Yaskawa INFORM job: KRIS1(-160_-90)07.JBI

/JOB
//NAME KRIS1(-160_-90)07
//POS
///NPOS 270,270,270,15,0,0
///TOOL 0
///POSTYPE PULSE
///PULSE
C00000=1357,-104031,-113776,-9484,62521,-80538
C00001=1357,-104031,-113776,-9484,62521,-80538
C00002=36470,-76528,-106815,-19279,71473,-77234
C00003=134470,-76528,-106815,-19279,71473,-77234
C00004=174981,-50493,-90161,-40064,84672,-66854
C00005=187879,-63712,-94262,-49080,81916,-61249
C00006=186060,-71155,-91964,-59790,82905,-66762
C00007=178869,-72848,-88692,-57971,77164,-66872
C00008=178869,-73293,-87273,-58169,76560,-66435
C00009=178869,-73560,-86246,-58315,76140,-66130
C00010=178674,-73111,-86205,-58218,76137,-66246
C00011=177360,-70267,-84836,-57702,75706,-66732
C00012=178674,-73111,-86205,-58218,76137,-66246
C00013=178674,-71838,-89995,-57689,77779,-67427
C00014=187879,-63712,-94262,-49080,81916,-61249
C00015=188382,-49930,-83952,-49213,82654,-61403
C00016=188014,-50962,-81654,-49243,81175,-60803
C00017=188014,-51673,-80691,-49342,80537,-60470
C00018=188014,-51583,-80818,-49329,80620,-60513
C00019=186548,-48975,-79328,-48719,80176,-60967
C00020=188014,-51583,-80818,-49329,80620,-60513
C00021=188014,-47372,-85350,-48920,83933,-62231
C00022=182062,-62332,-92296,-30199,64588,-50507
C00023=184090,-61700,-84500,-30217,57788,-46513
C00024=184090,-62275,-83323,-30540,56902,-46238
C00025=184090,-62207,-83473,-30499,57013,-46272
C00026=182547,-59219,-81900,-29317,56990,-46927
C00027=184090,-62207,-83473,-30499,57013,-46272
C00028=182062,-62332,-92296,-30199,64588,-50507
C00029=213458,-81436,-127572,-45024,85737,-46387
C00030=213462,-137262,-127618,-80891,60645,-46377
C00031=213462,-137262,-127618,-80891,60645,-46377
C00032=213462,-137262,-127281,-45256,60365,-46369
C00033=190178,-104312,-111371,-30656,55898,-55861
C00034=182510,-123951,-113302,-29184,45443,-56133
C00035=182510,-123446,-111392,-29630,44641,-55847
C00036=182510,-123495,-111565,-29589,44713,-55873
C00037=180510,-119420,-110276,-27514,45182,-57098
C00038=182510,-123495,-111565,-29589,44713,-55873
C00039=182510,-124409,-115363,-28705,46354,-56443
C00040=219776,-105077,-106077,-50090,64862,-45838
C00041=220601,-99189,-101769,-50266,65553,-45786
C00042=220601,-99263,-100237,-50600,64914,-45410
C00043=220601,-99258,-100424,-50559,64990,-45455
C00044=218392,-97957,-99927,-49618,64034,-46123
C00045=220601,-99258,-100424,-50559,64990,-45455
C00046=219776,-105077,-106077,-50090,64862,-45838
C00047=190178,-104312,-111371,-30656,55898,-55861
C00048=229240,-109114,-135810,-47014,82062,-49329
C00049=229240,-109114,-135810,-47014,82062,-49329
C00050=195224,-66819,-119592,-28790,78815,-60275
C00051=159578,-94739,-111578,-14965,102577,-71346
C00052=157566,-87256,-71357,-3912,80960,-68626
C00053=158237,-87274,-67249,-3997,78461,-68317
C00054=158512,-86753,-64553,-4040,77085,-68177
C00055=158512,-85902,-62577,-4050,76306,-68151
C00056=159334,-88042,-63583,-4126,75872,-67853
C00057=159947,-89575,-64280,-4185,75546,-67628
C00058=158678,-86897,-63962,-4060,76658,-68106
C00059=158401,-87046,-65688,-4022,77628,-68233
C00060=157724,-87159,-69865,-3934,80101,-68545
C00061=157573,-90681,-89077,-3900,90084,-68907
C00062=157703,-92030,-92713,-3898,91631,-68910
C00063=158377,-93978,-89476,-3949,88678,-68591
C00064=158653,-94353,-86922,-3974,86930,-68442
C00065=158653,-94065,-85585,-3975,86257,-68419
C00066=158901,-94897,-86117,-3998,86172,-68332
C00067=159738,-97484,-87119,-4071,85502,-68025
C00068=158508,-94414,-86637,-3961,86718,-68485
C00069=158233,-93872,-88035,-3937,87841,-68614
C00070=157561,-92106,-91348,-3883,90748,-68930
C00071=157550,-88189,-103730,-3988,100358,-69239
C00072=157494,-88262,-105997,-3987,101710,-69297
C00073=158163,-92718,-103752,-3992,98079,-68960
C00074=158927,-96366,-102620,-4029,95553,-68625
C00075=158927,-96520,-101690,-4026,94903,-68601
C00076=158927,-96495,-101852,-4026,95015,-68605
C00077=159979,-100458,-103367,-4107,93966,-68220
C00078=158702,-95424,-101809,-4010,95525,-68699
C00079=158425,-94019,-102865,-4000,96880,-68834
C00080=157748,-89886,-105246,-3989,100429,-69172
C00081=156260,-82084,-105550,-20461,72444,-69801
C00082=137260,-84248,-120477,-10166,77039,-76482
C00083=137260,-138866,-133764,-10166,31487,-76482
C00084=72641,-154229,-133982,-11252,19318,-75992
C00085=56453,-149109,-122299,-13274,13706,-75060
C00086=30023,-158112,-125301,-6799,9035,-78029
C00087=-11401,-148032,-125425,-11667,35640,-75771
C00088=-126225,-114648,-117375,-36487,17100,-65054
C00089=-160935,-140983,-109640,-13468,75088,-74332
C00090=-169853,-118963,-84593,-12681,69660,86771
C00091=-185015,-85467,-64977,-10138,72568,81037
C00092=-186046,-86587,-63372,-10054,70902,80807
C00093=-186046,-85672,-61299,-10100,70108,80875
C00094=-186099,-85805,-61481,-10085,70145,80849
C00095=-187639,-87511,-62050,-9863,69435,80354
C00096=-183812,-88241,-67244,-10331,72692,81455
C00097=-173907,-109296,-96285,-11524,80966,84205
C00098=-165243,-81442,-84446,-9619,88683,83239
C00099=-165243,-81286,-81084,-9622,86723,83389
C00100=-165344,-81527,-80785,-9608,86408,83377
C00101=-165344,-81401,-79599,-9612,85752,83428
C00102=-165344,-81434,-79892,-9611,85913,83415
C00103=-166373,-84175,-81092,-9484,85132,83124
C00104=-163979,-82682,-81772,-9785,86585,83830
C00105=-160654,-84295,-101618,-10197,98198,83833
C00106=-158831,-94543,-102742,-7696,93888,81952
C00107=-159073,-94488,-101668,-7659,93239,81911
C00108=-159073,-94700,-100523,-7653,92432,81960
C00109=-159073,-94669,-100714,-7655,92565,81952
C00110=-160071,-98397,-102165,-7522,91459,81686
C00111=-158831,-94357,-103427,-7703,94400,81921
C00112=-161715,-86803,-103327,-4886,98608,77730
C00113=-162141,-92472,-85533,3463,86932,68770
C00114=-161818,-87798,-71417,3733,80713,68419
C00115=-160875,-83714,-65601,3665,79192,68698
C00116=-161375,-83882,-63363,3725,77755,68482
C00117=-161375,-83186,-61665,3733,77069,68462
C00118=-161375,-83302,-61946,3731,77181,68466
C00119=-162606,-86103,-62964,3849,76427,68017
C00120=-161375,-84160,-64056,3722,78038,68491
C00121=-162005,-87841,-70029,3758,79847,68329
C00122=-161949,-92223,-96357,3744,93768,68761
C00123=-161804,-92637,-92737,3704,91325,68737
C00124=-160782,-89227,-87327,3611,89709,69033
C00125=-161425,-90912,-85851,3665,87970,68764
C00126=-161425,-90690,-84578,3665,87303,68744
C00127=-161425,-90728,-84781,3665,87408,68747
C00128=-162412,-93603,-85938,3751,86691,68391
C00129=-161425,-91016,-86520,3665,88326,68774
C00130=-162058,-93372,-91608,3722,90267,68620
C00131=-162002,-88104,-107646,3859,102814,69021
C00132=-161873,-89540,-106233,3806,101205,69011
C00133=-162580,-93883,-103932,3818,97597,68666
C00134=-159915,-93477,-102438,3577,96772,69526
C00135=-159915,-93839,-100899,3567,95642,69493
C00136=-159915,-93799,-101099,3568,95785,69497
C00137=-160794,-97042,-102371,3639,94941,69180
C00138=-159915,-93165,-103472,3585,97568,69550
C00139=-164885,-102201,-108421,4002,96197,67859
C00140=-149595,-96211,-103761,5489,101844,74102
C00141=-148895,-100989,-103442,6283,96942,74202
C00142=-149006,-93113,-100988,5479,101691,74295
C00143=-149599,-96300,-103483,5484,101628,74092
C00144=-137295,-108190,-106060,5698,94014,77976
C00145=-149608,-96287,-103789,5489,101823,74097
C00146=-160720,-151449,-123129,13814,72249,68439
C00147=-174899,-138237,-126795,-1008,88740,67536
C00148=-163022,-96341,-102515,-22398,105363,76518
C00149=-163017,-96713,-99258,-22147,103326,76913
C00150=-166118,-105377,-102170,-18852,96347,77230
C00151=-163022,-96736,-99152,-22139,103253,76925
C00152=-162158,-93804,-96763,-22109,103515,77196
C00153=-174925,-92085,-97088,-18785,97864,73864
C00154=-167549,-101389,-103915,-18999,98984,76305
C00155=-163194,-119427,-113025,-19710,97619,78016
C00156=-163006,-95534,-87485,-21597,97146,78065
C00157=-166449,-103981,-88986,-17839,88165,78380
C00158=-167279,-118842,-91930,-16839,77497,71410
C00159=-163006,-94576,-83573,-21494,95359,78388
C00160=-162142,-91714,-81191,-21448,95589,78662
C00161=-178049,-105864,-87645,-15594,79224,67328
C00162=-171906,-113065,-93299,-16245,80217,69386
C00163=-173072,-122981,-101575,4997,88706,65554
C00164=-166636,-106884,-92426,2568,94448,67910
C00165=-167630,-109607,-91139,2502,92292,67531
C00166=-162194,-92631,-84353,-657,102863,69400
C00167=-163060,-95514,-86735,-782,102839,69097
C00168=-155875,-120106,-94474,3152,88541,71437
C00169=-155875,-121766,-97691,3153,89666,71465
C00170=-178442,-133591,-104623,8068,82135,63325
C00171=-176542,-133362,-109369,6755,86992,64211
C00172=-163036,-88875,-67291,-2288,96831,69180
C00173=-159610,-85618,-62441,-1680,95605,70370
C00174=-162086,-85813,-60042,-2106,93969,69554
C00175=-162173,-84225,-60457,-2128,95039,69506
C00176=-163038,-86971,-62872,-2279,95091,69211
C00177=-151835,-92381,-62525,-304,92274,73022
C00178=-151835,-95702,-69255,-305,94709,73016
C00179=-163041,-94022,-81579,-12660,98605,75478
C00180=-162985,-87715,-64806,-21312,87868,79725
C00181=-162980,-85781,-60474,-21324,86307,80003
C00182=-163244,-83528,-57038,-21357,85347,80079
C00183=-162985,-85725,-60330,-21325,86250,80011
C00184=-162122,-82990,-57905,-21265,86391,80297
C00185=-171549,-75890,-53739,-21771,84944,77151
C00186=-153122,-94015,-66237,-20488,88162,83220
C00187=-168603,-127327,-105850,-12339,78437,-77405
C00188=-149894,-144724,-110594,-14594,75698,-70467
C00189=-126225,-114648,-117375,-36487,17100,-65054
C00190=-118781,-153853,-134406,-32592,23357,-65054
C00191=-12470,-167083,-125425,-11667,16324,-75771
C00192=137258,-84249,-120477,-10166,64820,-76482
C00193=160540,-100857,-113063,-23155,68829,-67581
C00194=174981,-50493,-90161,-40064,84672,-66854
C00195=187879,-63712,-94262,-49080,81916,-61249
C00196=230671,-89591,-126680,-64018,108053,-56526
C00197=230671,-150117,-126680,-83924,107200,-56526
C00198=230671,-150117,-126680,-83924,107200,-56526
C00199=230671,-150117,-126680,-39809,88276,-56526
C00200=185677,-128245,-133585,-38839,68006,-71149
C00201=143279,-154007,-127386,-2438,36675,-82296
C00202=143641,-141701,-120251,-2678,38614,-82167
C00203=143742,-142485,-120562,-2786,38406,-82105
C00204=143590,-141570,-120589,-2614,38886,-82201
C00205=202481,-119765,-113580,-40189,62069,-59692
C00206=198646,-130340,-109614,-41067,39992,-50520
C00207=196873,-131559,-103686,-47690,28279,-43258
C00208=193242,-140218,-107458,-47365,24899,-43542
C00209=143279,-154007,-127386,-2438,36675,-82296
C00210=143372,-162538,-136969,-2444,38193,-82294
C00211=143372,-162538,-136969,-2444,38193,-82294
C00212=169193,-120980,-126540,-32650,66176,-77929
C00213=162706,-113692,-115443,-30259,61179,-79142
C00214=159752,-104020,-109361,-28408,61247,-80415
C00215=143742,-142485,-120562,-2786,38406,-82105
C00216=143590,-141570,-120589,-2614,38886,-82201
C00217=133258,-125438,-116737,-13449,48460,-89137
C00218=140125,-121566,-112050,-33225,52073,-88232
C00219=147500,-115752,-104174,-50028,56665,-87600
C00220=148531,-114571,-100134,-56979,57308,-87783
C00221=151078,-112408,-101145,-56872,59820,-87990
C00222=162706,-113692,-115443,-30259,61179,-79142
C00223=169193,-120980,-126540,-32650,66176,-77929
C00224=169193,-120980,-126540,-32650,66176,-77929
C00225=169193,-120980,-126540,-32650,66176,-77929
C00226=169193,-120980,-126540,-32650,66176,-77929
C00227=189746,-144194,-133392,-42604,68859,-69788
C00228=182215,-131283,-122466,-40105,65254,-71827
C00229=178274,-121415,-115340,-38427,64020,-73174
C00230=157461,-154213,-124395,-33339,46072,-76518
C00231=155749,-154222,-121631,-44079,49487,-78540
C00232=159534,-158630,-125101,-47522,52653,-77846
C00233=179897,-166210,-133900,-51769,64813,-73191
C00234=179897,-166210,-133900,-51769,64813,-73191
C00235=179897,-166210,-133900,-51769,64813,-73191
C00236=144017,-127352,-123370,-33815,56946,-88116
C00237=136296,-120281,-120593,4079,55650,-85264
C00238=135299,-107675,-113640,4618,57894,-85562
C00239=145232,-101484,-111409,-1707,59530,-81793
C00240=158760,-87446,-105850,-9753,64232,-77140
C00241=147394,-98337,-102183,17301,47751,-78343
C00242=144875,-102905,-108473,14295,50590,-79740
C00243=136296,-120281,-120593,4079,55650,-85264
C00244=138675,-113827,-131364,2561,67962,-83610
C00245=184171,-107868,-119248,-16468,98370,-62097
C00246=171634,-136713,-119987,-14813,82155,-64373
C00247=159470,-98078,-104776,-5796,102446,-69552
C00248=161378,-95420,-100865,-5759,101546,-68862
C00249=158743,-95268,-103371,-5812,102972,-69826
C00250=157888,-92366,-100981,-5813,102933,-70115
C00251=150653,-106168,-104972,-5675,97814,-72341
C00252=153886,-106740,-107354,-5718,99208,-71304
C00253=163031,-143044,-118600,-5591,88166,-67691
C00254=166711,-113552,-95038,-4166,94777,-66107
C00255=166288,-102352,-87247,-1195,97977,-66532
C00256=158755,-94787,-86481,976,103949,-69303
C00257=157900,-91912,-84097,841,103969,-69603
C00258=155716,-111746,-90511,-2417,94923,-70111
C00259=153517,-115912,-96262,-2679,96250,-70891
C00260=166250,-149525,-105399,-1185,84912,-66421
C00261=160517,-92560,-68375,-1999,97708,-69937
C00262=161332,-84623,-58779,-1824,95900,-69631
C00263=158782,-86330,-62292,-2348,97119,-70521
C00264=157926,-83586,-59872,-2521,97014,-70811
C00265=150683,-91270,-61306,-3946,93662,-73181
C00266=149643,-98229,-74267,-4194,97999,-73676
C00267=159578,-94739,-111578,-14965,102577,-71346
C00268=134470,-76528,-106815,-19279,71473,-77234
C00269=36470,-76528,-106815,-19279,71473,-77234
BC00000=230661,511423,1075115
BC00001=230661,511423,1075115
BC00002=295309,515546,1075139
BC00003=353519,294132,1075139
BC00004=353008,251675,1075139
BC00005=352559,214443,1075139
BC00006=352563,214698,1075132
BC00007=352563,214698,1075132
BC00008=352563,214698,1075132
BC00009=352563,214698,1075132
BC00010=352563,214698,1075132
BC00011=352563,214698,1075132
BC00012=352563,214698,1075132
BC00013=352563,214698,1075132
BC00014=352559,214443,1075139
BC00015=352559,214443,1075139
BC00016=352559,214443,1075139
BC00017=352559,214443,1075139
BC00018=352559,214443,1075139
BC00019=352559,214443,1075136
BC00020=352559,214443,1075139
BC00021=352559,214443,1075139
BC00022=352559,214443,1075135
BC00023=352559,214443,1075135
BC00024=352559,214443,1075135
BC00025=352559,214443,1075135
BC00026=352559,214443,1075135
BC00027=352559,214443,1075135
BC00028=352559,214443,1075135
BC00029=352559,214443,1075135
BC00030=352559,214443,1075135
BC00031=265654,200751,1075135
BC00032=265654,200751,1075135
BC00033=265654,182191,1075135
BC00034=265654,182191,1075135
BC00035=265654,182191,1075135
BC00036=265654,182191,1075135
BC00037=265654,182191,1075135
BC00038=265654,182191,1075135
BC00039=265654,182191,1075135
BC00040=265654,153562,1075135
BC00041=265654,153562,1075135
BC00042=265654,153562,1075135
BC00043=265654,153562,1075135
BC00044=265654,153562,1075135
BC00045=265654,153562,1075135
BC00046=265654,153562,1075135
BC00047=265654,182191,1075135
BC00048=288097,183452,1075134
BC00049=288097,183452,1075134
BC00050=366407,228141,1075134
BC00051=353519,214242,1075139
BC00052=382934,213120,1075139
BC00053=382934,213120,1075139
BC00054=382934,213120,1075139
BC00055=382934,213120,1075139
BC00056=382933,213121,1075138
BC00057=382933,213121,1075138
BC00058=382934,213120,1075139
BC00059=382934,213120,1075139
BC00060=382934,213120,1075139
BC00061=382615,202068,1075139
BC00062=382076,183746,1075139
BC00063=382076,183746,1075139
BC00064=382076,183746,1075139
BC00065=382076,183746,1075139
BC00066=382076,183746,1075139
BC00067=382076,183746,1075139
BC00068=382076,183746,1075139
BC00069=382076,183746,1075139
BC00070=382076,183746,1075139
BC00071=382031,172700,1075139
BC00072=382054,156718,1075139
BC00073=382054,156718,1075139
BC00074=382054,156718,1075139
BC00075=382054,156718,1075139
BC00076=382054,156718,1075139
BC00077=382054,156718,1075139
BC00078=382054,156718,1075139
BC00079=382054,156718,1075139
BC00080=382054,156718,1075139
BC00081=381880,223521,1075139
BC00082=353800,266120,1075139
BC00083=353800,266120,1075139
BC00084=369629,142690,1075139
BC00085=373603,111702,1075139
BC00086=379757,63718,1075139
BC00087=398174,159824,1075139
BC00088=312616,52052,1075139
BC00089=340737,74809,1075139
BC00090=340750,75261,1075139
BC00091=340750,75261,1075139
BC00092=340750,75261,1075139
BC00093=340750,75261,1075139
BC00094=340750,75261,1075139
BC00095=340750,75261,1075139
BC00096=340750,75261,1075139
BC00097=340750,75261,1075139
BC00098=322858,75822,1075139
BC00099=322858,75822,1075139
BC00100=322858,75822,1075139
BC00101=322858,75822,1075139
BC00102=322858,75822,1075139
BC00103=322858,75822,1075139
BC00104=322858,75822,1075139
BC00105=321852,75909,1075139
BC00106=305307,104079,1075139
BC00107=305307,104079,1075139
BC00108=305307,104079,1075139
BC00109=305307,104079,1075139
BC00110=305307,104079,1075139
BC00111=305307,104079,1075139
BC00112=323389,89421,1075139
BC00113=381448,44122,1075139
BC00114=383279,43102,1075139
BC00115=383279,43102,1075139
BC00116=383279,43102,1075139
BC00117=383279,43102,1075139
BC00118=383279,43102,1075139
BC00119=383279,43102,1075139
BC00120=383279,43102,1075139
BC00121=383279,43102,1075139
BC00122=383346,62866,1075139
BC00123=383236,72913,1075139
BC00124=383236,72913,1075139
BC00125=383236,72913,1075139
BC00126=383236,72913,1075139
BC00127=383236,72913,1075139
BC00128=383236,72913,1075139
BC00129=383236,72913,1075139
BC00130=383236,72913,1075139
BC00131=383192,91135,1075139
BC00132=383033,99727,1075139
BC00133=383033,99727,1075139
BC00134=383033,99727,1075139
BC00135=383033,99727,1075139
BC00136=383033,99727,1075139
BC00137=383033,99727,1075139
BC00138=383033,99727,1075139
BC00139=383033,99727,1075139
BC00140=348621,100905,1075139
BC00141=348896,99875,1075139
BC00142=348896,99875,1075139
BC00143=348896,99875,1075139
BC00144=348896,99875,1075139
BC00145=364549,100867,1075139
BC00146=363863,103441,1075139
BC00147=346080,121643,1075139
BC00148=323509,144746,1075139
BC00149=322803,140398,1075139
BC00150=322592,139099,1075139
BC00151=322520,138659,1075139
BC00152=322520,138659,1075139
BC00153=322592,139099,1075139
BC00154=322592,139099,1075139
BC00155=318216,140757,1075139
BC00156=323435,117945,1075139
BC00157=322729,113597,1075139
BC00158=322729,113597,1075139
BC00159=322446,111858,1075139
BC00160=322446,111858,1075139
BC00161=322729,113597,1075139
BC00162=322729,113597,1075139
BC00163=364623,109054,1075139
BC00164=365306,105037,1075139
BC00165=365306,105037,1075139
BC00166=365579,103431,1075139
BC00167=365579,103431,1075139
BC00168=365306,105037,1075139
BC00169=365306,105037,1075139
BC00170=380551,109015,1075139
BC00171=378551,106052,1075139
BC00172=364555,85312,1075139
BC00173=365237,80960,1075139
BC00174=365237,80960,1075139
BC00175=365509,79219,1075139
BC00176=365509,79219,1075139
BC00177=365237,80960,1075139
BC00178=365237,80960,1075139
BC00179=341067,86785,1075139
BC00180=323352,88165,1075139
BC00181=322645,83817,1075139
BC00182=322645,83817,1075139
BC00183=322363,82077,1075139
BC00184=322363,82077,1075139
BC00185=322645,83817,1075139
BC00186=306969,83854,1075139
BC00187=340737,74809,1075139
BC00188=340737,74809,1075139
BC00189=312616,52052,1075139
BC00190=312616,52052,1075139
BC00191=398174,159824,1075139
BC00192=353801,266119,1075139
BC00193=381880,223521,1075139
BC00194=353008,251675,1075139
BC00195=352559,214443,1075139
BC00196=352559,214443,1075139
BC00197=269474,214443,1075139
BC00198=209500,192764,1075139
BC00199=229937,192764,1075139
BC00200=209500,192764,1075139
BC00201=209500,192764,1075139
BC00202=209500,192764,1075135
BC00203=209500,192764,1075135
BC00204=209500,192764,1075135
BC00205=234557,161453,1075132
BC00206=234557,161453,1075132
BC00207=234557,161453,1075132
BC00208=234557,161453,1075132
BC00209=209500,192764,1075139
BC00210=209501,302299,1075135
BC00211=304046,302299,1075135
BC00212=304046,203195,1075135
BC00213=304046,203195,1075135
BC00214=304046,203195,1075135
BC00215=209500,192764,1075135
BC00216=209500,192764,1075135
BC00217=304046,203195,1075135
BC00218=304046,203195,1075135
BC00219=304046,203195,1075135
BC00220=304046,203195,1075135
BC00221=304046,203195,1075135
BC00222=304046,203195,1075135
BC00223=304046,203195,1075135
BC00224=304046,310775,1075135
BC00225=206063,312405,1075135
BC00226=206063,203684,1075135
BC00227=216899,182662,1075135
BC00228=216899,182662,1075135
BC00229=216899,182662,1075135
BC00230=216899,182662,1075135
BC00231=216898,182663,1075134
BC00232=216899,182662,1075135
BC00233=216898,182662,1075132
BC00234=216898,281603,1075132
BC00235=299601,281603,1075132
BC00236=274761,236253,1075132
BC00237=304046,203195,1075135
BC00238=304046,203195,1075135
BC00239=304046,203195,1075135
BC00240=304045,203195,1075131
BC00241=304046,203195,1075135
BC00242=304046,203195,1075135
BC00243=304046,203195,1075135
BC00244=308056,199315,1075135
BC00245=363620,145544,1075139
BC00246=363620,145544,1075139
BC00247=364348,148086,1075139
BC00248=364638,149103,1075136
BC00249=364639,149103,1075139
BC00250=364639,149103,1075139
BC00251=364638,149103,1075136
BC00252=370099,148733,1075137
BC00253=370099,148733,1075137
BC00254=364145,147610,1075137
BC00255=364418,149141,1075138
BC00256=364758,151053,1075139
BC00257=364758,151053,1075139
BC00258=364418,149141,1075138
BC00259=364418,149141,1075138
BC00260=364418,149141,1075138
BC00261=353519,171684,1075139
BC00262=355504,177664,1075139
BC00263=355504,177664,1075139
BC00264=355504,177664,1075139
BC00265=355504,177664,1075139
BC00266=355504,177664,1075139
BC00267=353519,214242,1075139
BC00268=353519,294132,1075139
BC00269=295309,515546,1075139
EC00000=-12352,-159808
EC00001=1418783,-184756
EC00002=1418945,372643
EC00003=1418945,372643
EC00004=1342906,372643
EC00005=1276223,372643
EC00006=1276676,372643
EC00007=1276676,372643
EC00008=1276676,372643
EC00009=1276676,372643
EC00010=1276676,372643
EC00011=1276676,372643
EC00012=1276676,372643
EC00013=1276676,372643
EC00014=1276223,372643
EC00015=1276223,372643
EC00016=1276223,372643
EC00017=1276223,372643
EC00018=1276223,372643
EC00019=1276222,372643
EC00020=1276223,372643
EC00021=1276223,372643
EC00022=1276222,372644
EC00023=1276222,372644
EC00024=1276222,372644
EC00025=1276222,372644
EC00026=1276222,372644
EC00027=1276222,372644
EC00028=1276222,372644
EC00029=1276222,372644
EC00030=1276222,372644
EC00031=1276222,372644
EC00032=1276222,372644
EC00033=1276222,372644
EC00034=1276222,372644
EC00035=1276222,372644
EC00036=1276222,372644
EC00037=1276222,372644
EC00038=1276222,372644
EC00039=1276222,372644
EC00040=1276222,372644
EC00041=1276222,372644
EC00042=1276222,372644
EC00043=1276222,372644
EC00044=1276222,372644
EC00045=1276222,372644
EC00046=1276222,372644
EC00047=1276222,372644
EC00048=1276222,372644
EC00049=1276222,372644
EC00050=1276222,372644
EC00051=1418945,372643
EC00052=1418945,372643
EC00053=1418945,372643
EC00054=1418945,372643
EC00055=1418945,372643
EC00056=1418943,372643
EC00057=1418943,372643
EC00058=1418945,372643
EC00059=1418945,372643
EC00060=1418945,372643
EC00061=1418945,372643
EC00062=1418945,372643
EC00063=1418945,372643
EC00064=1418945,372643
EC00065=1418945,372643
EC00066=1418945,372643
EC00067=1418945,372643
EC00068=1418945,372643
EC00069=1418945,372643
EC00070=1418945,372643
EC00071=1418945,372643
EC00072=1418945,372643
EC00073=1418945,372643
EC00074=1418945,372643
EC00075=1418945,372643
EC00076=1418945,372643
EC00077=1418945,372643
EC00078=1418945,372643
EC00079=1418945,372643
EC00080=1418945,372643
EC00081=1418945,372643
EC00082=1418945,372643
EC00083=1418945,372643
EC00084=1418945,372643
EC00085=1418945,372643
EC00086=1418945,372643
EC00087=1595090,-179995
EC00088=1773681,-740307
EC00089=1773681,-740307
EC00090=1773681,-740307
EC00091=1773681,-740307
EC00092=1773681,-740307
EC00093=1773681,-740307
EC00094=1773681,-740307
EC00095=1773681,-740307
EC00096=1773681,-740307
EC00097=1773681,-740307
EC00098=1773681,-740307
EC00099=1773681,-740307
EC00100=1773681,-740307
EC00101=1773681,-740307
EC00102=1773681,-740307
EC00103=1773681,-740307
EC00104=1773681,-740307
EC00105=1773681,-740307
EC00106=1773681,-740307
EC00107=1773681,-740307
EC00108=1773681,-740307
EC00109=1773681,-740307
EC00110=1773681,-740307
EC00111=1773681,-740307
EC00112=1773681,-740307
EC00113=1773681,-740307
EC00114=1773681,-740307
EC00115=1773681,-740307
EC00116=1773681,-740307
EC00117=1773681,-740307
EC00118=1773681,-740307
EC00119=1773681,-740307
EC00120=1773681,-740307
EC00121=1773681,-740307
EC00122=1773681,-740307
EC00123=1773681,-740307
EC00124=1773681,-740307
EC00125=1773681,-740307
EC00126=1773681,-740307
EC00127=1773681,-740307
EC00128=1773681,-740307
EC00129=1773681,-740307
EC00130=1773681,-740307
EC00131=1773681,-740307
EC00132=1773681,-740307
EC00133=1773681,-740307
EC00134=1773681,-740307
EC00135=1773681,-740307
EC00136=1773681,-740307
EC00137=1773681,-740307
EC00138=1773681,-740307
EC00139=1773681,-740307
EC00140=1773681,-740307
EC00141=1773681,-740307
EC00142=1773681,-740307
EC00143=1773681,-740307
EC00144=1773681,-740307
EC00145=1773681,-740307
EC00146=1773681,-740307
EC00147=1773681,-740307
EC00148=1773681,-740307
EC00149=1773681,-740307
EC00150=1773681,-740307
EC00151=1773681,-740307
EC00152=1773681,-740307
EC00153=1773681,-740307
EC00154=1773681,-740307
EC00155=1773681,-740307
EC00156=1773681,-740307
EC00157=1773681,-740307
EC00158=1773681,-740307
EC00159=1773681,-740307
EC00160=1773681,-740307
EC00161=1773681,-740307
EC00162=1773681,-740307
EC00163=1773681,-740307
EC00164=1773681,-740307
EC00165=1773681,-740307
EC00166=1773681,-740307
EC00167=1773681,-740307
EC00168=1773681,-740307
EC00169=1773681,-740307
EC00170=1773681,-740307
EC00171=1773681,-740307
EC00172=1773681,-740307
EC00173=1773681,-740307
EC00174=1773681,-740307
EC00175=1773681,-740307
EC00176=1773681,-740307
EC00177=1773681,-740307
EC00178=1773681,-740307
EC00179=1773681,-740307
EC00180=1773681,-740307
EC00181=1773681,-740307
EC00182=1773681,-740307
EC00183=1773681,-740307
EC00184=1773681,-740307
EC00185=1773681,-740307
EC00186=1773681,-740307
EC00187=1773681,-740307
EC00188=1773681,-740307
EC00189=1773681,-740307
EC00190=1773681,-740307
EC00191=1595090,-179995
EC00192=1418947,372636
EC00193=1418945,372643
EC00194=1342906,372643
EC00195=1276223,372643
EC00196=1276223,372643
EC00197=1276223,372643
EC00198=1276223,372643
EC00199=1276223,372643
EC00200=1276223,372643
EC00201=1276223,372643
EC00202=1276222,372643
EC00203=1276222,372643
EC00204=1276222,372643
EC00205=1276221,372643
EC00206=1276221,372643
EC00207=1276221,372643
EC00208=1276221,372643
EC00209=1276223,372643
EC00210=1276222,372643
EC00211=1276222,372643
EC00212=1276222,372643
EC00213=1276222,372643
EC00214=1276222,372643
EC00215=1276222,372643
EC00216=1276222,372643
EC00217=1276222,372643
EC00218=1276222,372643
EC00219=1276222,372643
EC00220=1276222,372643
EC00221=1276222,372643
EC00222=1276222,372643
EC00223=1276222,372643
EC00224=1276222,372643
EC00225=1276222,372643
EC00226=1276222,372643
EC00227=1276222,372643
EC00228=1276222,372643
EC00229=1276222,372643
EC00230=1276222,372643
EC00231=1276221,372644
EC00232=1276222,372643
EC00233=1276221,372643
EC00234=1276221,372643
EC00235=1276221,372643
EC00236=1276221,372643
EC00237=1276222,372643
EC00238=1276222,372643
EC00239=1276222,372643
EC00240=1276222,372644
EC00241=1276222,372643
EC00242=1276222,372643
EC00243=1276222,372643
EC00244=1285829,372643
EC00245=1418945,372643
EC00246=1418945,372643
EC00247=1418945,372643
EC00248=1418945,372643
EC00249=1418945,372643
EC00250=1418945,372643
EC00251=1418945,372643
EC00252=1418945,372643
EC00253=1418945,372643
EC00254=1418944,372643
EC00255=1418944,372643
EC00256=1418945,372643
EC00257=1418945,372643
EC00258=1418944,372643
EC00259=1418944,372643
EC00260=1418944,372643
EC00261=1418945,372643
EC00262=1418945,372643
EC00263=1418945,372643
EC00264=1418945,372643
EC00265=1418945,372643
EC00266=1418945,372643
EC00267=1418945,372643
EC00268=1418945,372643
EC00269=1418945,372643
///POSTYPE BASE
///RECTAN
///RCONF 0,0,0,0,1,0,0,0,0,0,0,0,0,0,0,0,0,0,0,0,0,0,0,0
P00006=2.006,1.622,-0.565,0.0000,0.0000,0.0000
P00021=0.073,2.058,-0.109,0.0000,0.0000,0.0000
P00022=2.006,1.622,-0.565,0.0000,0.0000,0.0000
///RCONF 0,0,0,0,0,0,0,0,0,0,0,0,0,0,0,0,0,0,0,0,0,0,0,0
P00023=-2.957,-4.083,2.762,0.0000,0.0000,0.0000
P00031=-0.170,0.039,-0.647,0.0000,0.0000,0.0000
P00032=-0.423,0.157,3.222,0.0000,0.0000,0.0000
P00033=0.854,-1.099,3.047,0.0000,0.0000,0.0000
///RCONF 0,0,0,0,1,0,0,0,0,0,0,0,0,0,0,0,0,0,0,0,0,0,0,0
P00034=-8.151,9.743,-4.393,0.0000,0.0000,0.0000
///RCONF 0,0,0,0,0,0,0,0,0,0,0,0,0,0,0,0,0,0,0,0,0,0,0,0
P00035=0.390,-0.027,1.040,0.0000,0.0000,0.0000
P00036=-2.434,0.084,0.197,0.0000,0.0000,0.0000
P00051=-5.945,4.696,-10.293,0.0000,0.0000,0.0000
P00052=-0.153,5.586,-7.982,0.0000,0.0000,0.0000
P00053=0.015,-0.644,-4.942,0.0000,0.0000,0.0000
P00054=-0.184,15.039,-0.270,0.0000,0.0000,0.0000
P00055=-0.009,2.790,-4.790,0.0000,0.0000,0.0000
//INST
///DATE 2024/11/18 15:49
///ATTR SC,RW
///GROUP1 RB1,BS1
///GROUP2 ST1
NOP
SFTOF
SSFTOF
SFTOF3D
'OK_r2_O7.1(P)(-160.-90)
MOVJ C00000 BC00000 VJ=100.00  +MOVJ EC00000 VJ=100.00
MOVJ C00001 BC00001 VJ=100.00  +MOVJ EC00001 VJ=100.00
MOVJ C00002 BC00002 VJ=100.00  +MOVJ EC00002 VJ=100.00
MOVJ C00003 BC00003 VJ=100.00  +MOVJ EC00003 VJ=100.00
MOVJ C00004 BC00004 VJ=50.00  +MOVJ EC00004 VJ=50.00
MOVJ C00005 BC00005 VJ=50.00  +MOVJ EC00005 VJ=50.00
'DODAC SEARCH NO NOWA SPOINE
MOVL C00006 BC00006 V=400.0  +MOVJ EC00006 VJ=100.00
SMOVL C00007 BC00007 V=400.0  +MOVJ EC00007
SFTOF3D
SMOVL C00008 BC00008 V=100.0  +MOVJ EC00008
SREFP 3 C00009 BC00009  +REFP EC00009
CALL JOB:SEARCH-R1-S13D
SET P051 P006
SFTON3D P051
SMOVL C00010 BC00010 V=100.0  +MOVJ EC00010
SREFP 3 C00011 BC00011  +REFP EC00011
CALL JOB:SEARCH-R1-S13D
SET P051 P006
SFTON3D P051
SMOVL C00012 BC00012 V=100.0  +MOVJ EC00012
MOVL C00013 BC00013 V=400.0  +MOVJ EC00013 VJ=100.00
MOVL C00014 BC00014 V=400.0  +MOVJ EC00014 VJ=100.00
SFTOF3D
MOVL C00015 BC00015 V=400.0  +MOVJ EC00015 VJ=100.00
SMOVL C00016 BC00016 V=100.0  +MOVJ EC00016
SREFP 3 C00017 BC00017  +REFP EC00017
CALL JOB:SEARCH-R1-S13D
SET P052 P006
SFTON3D P052
SMOVL C00018 BC00018 V=100.0  +MOVJ EC00018
SREFP 3 C00019 BC00019  +REFP EC00019
CALL JOB:SEARCH-R1-S13D
SET P052 P006
SFTON3D P052
SMOVL C00020 BC00020 V=100.0  +MOVJ EC00020
MOVL C00021 BC00021 V=400.0  +MOVJ EC00021 VJ=100.00
SFTOF3D
MOVL C00022 BC00022 V=400.0  +MOVJ EC00022 VJ=100.00
SMOVL C00023 BC00023 V=100.0  +MOVJ EC00023
SREFP 3 C00024 BC00024  +REFP EC00024
CALL JOB:SEARCH-R1-S13D
SET P053 P006
SFTON3D P053
SMOVL C00025 BC00025 V=100.0  +MOVJ EC00025
SREFP 3 C00026 BC00026  +REFP EC00026
CALL JOB:SEARCH-R1-S13D
SET P053 P006
SFTON3D P053
SMOVL C00027 BC00027 V=100.0  +MOVJ EC00027
MOVL C00028 BC00028 V=400.0  +MOVJ EC00028 VJ=100.00
SFTOF3D
MOVL C00029 BC00029 V=400.0  +MOVJ EC00029 VJ=100.00
MOVL C00030 BC00030 V=400.0  +MOVJ EC00030 VJ=100.00
MOVL C00031 BC00031 V=400.0  +MOVJ EC00031 VJ=100.00
MOVL C00032 BC00032 V=400.0  +MOVJ EC00032 VJ=100.00
SFTOF3D
MOVL C00033 BC00033 V=400.0  +MOVJ EC00033 VJ=100.00
SMOVL C00034 BC00034 V=100.0  +MOVJ EC00034
SREFP 3 C00035 BC00035  +REFP EC00035
CALL JOB:SEARCH-R1-S13D
SET P054 P006
SFTON3D P054
SMOVL C00036 BC00036 V=100.0  +MOVJ EC00036
SREFP 3 C00037 BC00037  +REFP EC00037
CALL JOB:SEARCH-R1-S13D
SET P054 P006
SFTON3D P054
SMOVL C00038 BC00038 V=100.0  +MOVJ EC00038
MOVL C00039 BC00039 V=400.0  +MOVJ EC00039 VJ=100.00
SFTOF3D
MOVL C00040 BC00040 V=400.0  +MOVJ EC00040 VJ=100.00
SMOVL C00041 BC00041 V=100.0  +MOVJ EC00041
SREFP 3 C00042 BC00042  +REFP EC00042
CALL JOB:SEARCH-R1-S13D
SET P055 P006
SFTON3D P055
SMOVL C00043 BC00043 V=100.0  +MOVJ EC00043
SREFP 3 C00044 BC00044  +REFP EC00044
CALL JOB:SEARCH-R1-S13D
SET P055 P006
SFTON3D P055
SMOVL C00045 BC00045 V=100.0  +MOVJ EC00045
MOVL C00046 BC00046 V=400.0  +MOVJ EC00046 VJ=100.00
SFTOF3D
MOVL C00047 BC00047 V=400.0  +MOVJ EC00047 VJ=100.00
MOVL C00048 BC00048 V=400.0  +MOVJ EC00048 VJ=100.00
MOVL C00049 BC00049 V=400.0  +MOVJ EC00049 VJ=100.00
MOVL C00050 BC00050 V=400.0  +MOVJ EC00050 VJ=100.00
MOVJ C00051 BC00051 VJ=100.00  +MOVJ EC00051 VJ=100.00
'Path S1422
SFTOF3D
MOVJ C00052 BC00052 VJ=100.00  +MOVJ EC00052 VJ=100.00
MOVL C00053 BC00053 V=400.0  +MOVJ EC00053 VJ=100.00
SMOVL C00054 BC00054 V=100.0  +MOVJ EC00054
SREFP 3 C00055 BC00055  +REFP EC00055
CALL JOB:SEARCH-R1-S13D
SET P021 P006
SFTON3D P021
SMOVL C00056 BC00056 V=100.0  +MOVJ EC00056
SREFP 3 C00057 BC00057  +REFP EC00057
CALL JOB:SEARCH-R1-S13D
SET P021 P006
SFTON3D P021
SMOVL C00058 BC00058 V=100.0  +MOVJ EC00058
MOVL C00059 BC00059 V=400.0  +MOVJ EC00059 VJ=100.00
MOVL C00060 BC00060 V=1000.0  +MOVJ EC00060 VJ=100.00
MOVJ C00061 BC00061 VJ=100.00  +MOVJ EC00061 VJ=100.00
'Path S1423
SFTOF3D
MOVJ C00062 BC00062 VJ=100.00  +MOVJ EC00062 VJ=100.00
MOVL C00063 BC00063 V=400.0  +MOVJ EC00063 VJ=100.00
SMOVL C00064 BC00064 V=100.0  +MOVJ EC00064
SREFP 3 C00065 BC00065  +REFP EC00065
CALL JOB:SEARCH-R1-S13D
SET P022 P006
SFTON3D P022
SMOVL C00066 BC00066 V=100.0  +MOVJ EC00066
SREFP 3 C00067 BC00067  +REFP EC00067
CALL JOB:SEARCH-R1-S13D
SET P022 P006
SFTON3D P022
SMOVL C00068 BC00068 V=100.0  +MOVJ EC00068
MOVL C00069 BC00069 V=400.0  +MOVJ EC00069 VJ=100.00
MOVL C00070 BC00070 V=1000.0  +MOVJ EC00070 VJ=100.00
MOVJ C00071 BC00071 VJ=100.00  +MOVJ EC00071 VJ=100.00
'Path S1424
SFTOF3D
MOVJ C00072 BC00072 VJ=100.00  +MOVJ EC00072 VJ=100.00
MOVL C00073 BC00073 V=400.0  +MOVJ EC00073 VJ=100.00
SMOVL C00074 BC00074 V=100.0  +MOVJ EC00074
SREFP 3 C00075 BC00075  +REFP EC00075
CALL JOB:SEARCH-R1-S13D
SET P023 P006
SFTON3D P023
SMOVL C00076 BC00076 V=100.0  +MOVJ EC00076
SREFP 3 C00077 BC00077  +REFP EC00077
CALL JOB:SEARCH-R1-S13D
SET P023 P006
SFTON3D P023
SFTOF3D
SMOVL C00078 BC00078 V=100.0  +MOVJ EC00078
MOVL C00079 BC00079 V=400.0  +MOVJ EC00079 VJ=100.00
MOVL C00080 BC00080 V=1000.0  +MOVJ EC00080 VJ=100.00
'obrot
MOVJ C00081 BC00081 VJ=100.00  +MOVJ EC00081 VJ=100.00
MOVJ C00082 BC00082 VJ=100.00  +MOVJ EC00082 VJ=100.00
MOVJ C00083 BC00083 VJ=100.00  +MOVJ EC00083 VJ=100.00
MOVJ C00084 BC00084 VJ=50.00  +MOVJ EC00084 VJ=50.00
MOVJ C00085 BC00085 VJ=50.00  +MOVJ EC00085 VJ=50.00
MOVJ C00086 BC00086 VJ=100.00  +MOVJ EC00086 VJ=100.00
MOVJ C00087 BC00087 VJ=100.00  +MOVJ EC00087 VJ=100.00
MOVJ C00088 BC00088 VJ=100.00  +MOVJ EC00088 VJ=100.00
MOVJ C00089 BC00089 VJ=100.00  +MOVJ EC00089 VJ=100.00
'Path S1077
SFTOF3D
MOVJ C00090 BC00090 VJ=100.00  +MOVJ EC00090 VJ=100.00
MOVL C00091 BC00091 V=400.0  +MOVJ EC00091 VJ=100.00
SMOVL C00092 BC00092 V=100.0  +MOVJ EC00092
SREFP 3 C00093 BC00093  +REFP EC00093
CALL JOB:SEARCH-R1-S13D
SET P031 P006
SFTON3D P031
SMOVL C00094 BC00094 V=100.0  +MOVJ EC00094
SREFP 3 C00095 BC00095  +REFP EC00095
CALL JOB:SEARCH-R1-S13D
SET P031 P006
SFTON3D P031
SMOVL C00096 BC00096 V=100.0  +MOVJ EC00096
MOVL C00097 BC00097 V=1000.0  +MOVJ EC00097 VJ=100.00
MOVJ C00098 BC00098 VJ=100.00  +MOVJ EC00098 VJ=100.00
'Path S1078
SFTOF3D
MOVL C00099 BC00099 V=400.0  +MOVJ EC00099 VJ=100.00
SMOVL C00100 BC00100 V=100.0  +MOVJ EC00100
SREFP 3 C00101 BC00101  +REFP EC00101
CALL JOB:SEARCH-R1-S13D
SET P032 P006
SFTON3D P032
SMOVL C00102 BC00102 V=100.0  +MOVJ EC00102
SREFP 3 C00103 BC00103  +REFP EC00103
CALL JOB:SEARCH-R1-S13D
SET P032 P006
SFTON3D P032
SMOVL C00104 BC00104 V=100.0  +MOVJ EC00104
MOVL C00105 BC00105 V=1000.0  +MOVJ EC00105 VJ=100.00
'Path S1079
SFTOF3D
MOVL C00106 BC00106 V=400.0  +MOVJ EC00106 VJ=100.00
SMOVL C00107 BC00107 V=100.0  +MOVJ EC00107
SREFP 3 C00108 BC00108  +REFP EC00108
CALL JOB:SEARCH-R1-S13D
SET P033 P006
SFTON3D P033
SMOVL C00109 BC00109 V=100.0  +MOVJ EC00109
SREFP 3 C00110 BC00110  +REFP EC00110
CALL JOB:SEARCH-R1-S13D
SET P033 P006
SFTON3D P033
SMOVL C00111 BC00111 V=100.0  +MOVJ EC00111
MOVJ C00112 BC00112 VJ=100.00  +MOVJ EC00112 VJ=100.00
MOVJ C00113 BC00113 VJ=100.00  +MOVJ EC00113 VJ=100.00
'Path S1080
SFTOF3D
MOVJ C00114 BC00114 VJ=100.00  +MOVJ EC00114 VJ=100.00
MOVL C00115 BC00115 V=400.0  +MOVJ EC00115 VJ=100.00
SMOVL C00116 BC00116 V=100.0  +MOVJ EC00116
SREFP 3 C00117 BC00117  +REFP EC00117
CALL JOB:SEARCH-R1-S13D
SET P034 P006
SFTON3D P034
SMOVL C00118 BC00118 V=100.0  +MOVJ EC00118
SREFP 3 C00119 BC00119  +REFP EC00119
CALL JOB:SEARCH-R1-S13D
SET P034 P006
SFTON3D P034
SMOVL C00120 BC00120 V=100.0  +MOVJ EC00120
MOVL C00121 BC00121 V=1000.0  +MOVJ EC00121 VJ=100.00
MOVJ C00122 BC00122 VJ=100.00  +MOVJ EC00122 VJ=100.00
'Path S1081
SFTOF3D
MOVJ C00123 BC00123 VJ=100.00  +MOVJ EC00123 VJ=100.00
MOVL C00124 BC00124 V=400.0  +MOVJ EC00124 VJ=100.00
SMOVL C00125 BC00125 V=100.0  +MOVJ EC00125
SREFP 3 C00126 BC00126  +REFP EC00126
CALL JOB:SEARCH-R1-S13D
SET P035 P006
SFTON3D P035
SMOVL C00127 BC00127 V=100.0  +MOVJ EC00127
SREFP 3 C00128 BC00128  +REFP EC00128
CALL JOB:SEARCH-R1-S13D
SET P035 P006
SFTON3D P035
SMOVL C00129 BC00129 V=100.0  +MOVJ EC00129
MOVL C00130 BC00130 V=1000.0  +MOVJ EC00130 VJ=100.00
MOVJ C00131 BC00131 VJ=100.00  +MOVJ EC00131 VJ=100.00
'Path S1082
SFTOF3D
MOVJ C00132 BC00132 VJ=100.00  +MOVJ EC00132 VJ=100.00
MOVL C00133 BC00133 V=400.0  +MOVJ EC00133 VJ=100.00
SMOVL C00134 BC00134 V=100.0  +MOVJ EC00134
SREFP 3 C00135 BC00135  +REFP EC00135
CALL JOB:SEARCH-R1-S13D
SET P036 P006
SFTON3D P036
SMOVL C00136 BC00136 V=100.0  +MOVJ EC00136
SREFP 3 C00137 BC00137  +REFP EC00137
CALL JOB:SEARCH-R1-S13D
SET P036 P006
SFTON3D P036
SMOVL C00138 BC00138 V=133.3  +MOVJ EC00138
MOVL C00139 BC00139 V=400.0  +MOVJ EC00139 VJ=100.00
'Path W260
SFTOF3D
SFTON3D P036
SMOVL C00140 BC00140 V=400.0  +MOVJ EC00140
SMOVL C00141 BC00141 V=166.7 PL=0  +MOVJ EC00141
SREFP 1 C00142 BC00142  +REFP EC00142
SREFP 2 C00143 BC00143  +REFP EC00143
MACRO1 MJ#(0) ARGF14
ARCON
SMOVL C00144 BC00144 V=10.0  +MOVJ EC00144
ARCOF
SMOVL C00145 BC00145 V=400.0  +MOVJ EC00145
SMOVL C00146 BC00146 V=1000.0  +MOVJ EC00146
SFTOF3D
MOVJ C00147 BC00147 VJ=100.00  +MOVJ EC00147 VJ=100.00
'Path W261
SFTOF3D
SFTON3D P033
MOVJ C00148 BC00148 VJ=100.00  +MOVJ EC00148 VJ=100.00
SMOVL C00149 BC00149 V=400.0  +MOVJ EC00149
SMOVL C00150 BC00150 V=133.3 PL=0  +MOVJ EC00150
SREFP 1 C00151 BC00151  +REFP EC00151
SREFP 2 C00152 BC00152  +REFP EC00152
MACRO1 MJ#(0) ARGF14
ARCON
SMOVL C00153 BC00153 V=10.0  +MOVJ EC00153
ARCOF
SMOVL C00154 BC00154 V=400.0  +MOVJ EC00154
SMOVL C00155 BC00155 V=1000.0  +MOVJ EC00155
SFTOF3D
'Path W1083
SFTOF3D
SFTON3D P032
MOVJ C00156 BC00156 VJ=100.00  +MOVJ EC00156 VJ=100.00
SMOVL C00157 BC00157 V=400.0  +MOVJ EC00157
SMOVL C00158 BC00158 V=133.3 PL=0  +MOVJ EC00158
SREFP 1 C00159 BC00159  +REFP EC00159
SREFP 2 C00160 BC00160  +REFP EC00160
MACRO1 MJ#(0) ARGF14
ARCON
SMOVL C00161 BC00161 V=10.0  +MOVJ EC00161
ARCOF
SMOVL C00162 BC00162 V=400.0  +MOVJ EC00162
SFTOF3D
'Path W262
SFTOF3D
SFTON3D P035
MOVJ C00163 BC00163 VJ=100.00  +MOVJ EC00163 VJ=100.00
SMOVL C00164 BC00164 V=400.0  +MOVJ EC00164
SMOVL C00165 BC00165 V=133.3 PL=0  +MOVJ EC00165
SREFP 1 C00166 BC00166  +REFP EC00166
SREFP 2 C00167 BC00167  +REFP EC00167
MACRO1 MJ#(0) ARGF14
ARCON
SMOVL C00168 BC00168 V=10.0  +MOVJ EC00168
ARCOF
SMOVL C00169 BC00169 V=400.0  +MOVJ EC00169
SMOVL C00170 BC00170 V=1000.0  +MOVJ EC00170
SFTOF3D
MOVJ C00171 BC00171 VJ=100.00  +MOVJ EC00171 VJ=100.00
'Path W264
SFTOF3D
SFTON3D P034
MOVJ C00172 BC00172 VJ=100.00  +MOVJ EC00172 VJ=100.00
SMOVL C00173 BC00173 V=400.0  +MOVJ EC00173
SMOVL C00174 BC00174 V=100.0 PL=0  +MOVJ EC00174
SREFP 1 C00175 BC00175  +REFP EC00175
SREFP 2 C00176 BC00176  +REFP EC00176
MACRO1 MJ#(0) ARGF14
ARCON
SMOVL C00177 BC00177 V=10.0  +MOVJ EC00177
ARCOF
SMOVL C00178 BC00178 V=400.0  +MOVJ EC00178
SFTOF3D
MOVJ C00179 BC00179 VJ=100.00  +MOVJ EC00179 VJ=100.00
'Path W263
SFTOF3D
SFTON3D P031
MOVJ C00180 BC00180 VJ=100.00  +MOVJ EC00180 VJ=100.00
SMOVL C00181 BC00181 V=400.0  +MOVJ EC00181
SMOVL C00182 BC00182 V=133.3 PL=0  +MOVJ EC00182
SREFP 1 C00183 BC00183  +REFP EC00183
SREFP 2 C00184 BC00184  +REFP EC00184
MACRO1 MJ#(0) ARGF14
ARCON
SMOVL C00185 BC00185 V=10.0  +MOVJ EC00185
ARCOF
SMOVL C00186 BC00186 V=400.0  +MOVJ EC00186
SFTOF3D
'obrot
MOVJ C00187 BC00187 VJ=100.00  +MOVJ EC00187 VJ=100.00
MOVJ C00188 BC00188 VJ=100.00  +MOVJ EC00188 VJ=100.00
MOVJ C00189 BC00189 VJ=100.00  +MOVJ EC00189 VJ=100.00
MOVJ C00190 BC00190 VJ=100.00  +MOVJ EC00190 VJ=100.00
MOVJ C00191 BC00191 VJ=100.00  +MOVJ EC00191 VJ=100.00
MOVJ C00192 BC00192 VJ=100.00  +MOVJ EC00192 VJ=100.00
MOVJ C00193 BC00193 VJ=100.00  +MOVJ EC00193 VJ=100.00
MOVJ C00194 BC00194 VJ=50.00  +MOVJ EC00194 VJ=50.00
MOVJ C00195 BC00195 VJ=50.00  +MOVJ EC00195 VJ=50.00
MOVL C00196 BC00196 V=400.0  +MOVJ EC00196 VJ=100.00
MOVL C00197 BC00197 V=400.0  +MOVJ EC00197 VJ=100.00
MOVL C00198 BC00198 V=400.0  +MOVJ EC00198 VJ=100.00
MOVL C00199 BC00199 V=400.0  +MOVJ EC00199 VJ=100.00
MOVL C00200 BC00200 V=400.0  +MOVJ EC00200 VJ=100.00
MOVL C00201 BC00201 V=400.0  +MOVJ EC00201 VJ=100.00
SFTON3D P054
SMOVL C00202 BC00202 V=133.3 PL=0  +MOVJ EC00202
SREFP 1 C00203 BC00203  +REFP EC00203
SREFP 2 C00204 BC00204  +REFP EC00204
MACRO1 MJ#(0) ARGF14
ARCON
SFTON3D P055
SMOVL C00205 BC00205 V=11.7  +MOVJ EC00205
SMOVL C00206 BC00206 V=11.7  +MOVJ EC00206
SMOVL C00207 BC00207 V=11.7  +MOVJ EC00207
ARCOF
SMOVL C00208 BC00208 V=166.7  +MOVJ EC00208
SMOVL C00209 BC00209 V=400.0  +MOVJ EC00209
SFTOF3D
SMOVL C00210 BC00210 V=400.0  +MOVJ EC00210
SMOVL C00211 BC00211 V=400.0  +MOVJ EC00211
SMOVL C00212 BC00212 V=400.0  +MOVJ EC00212
SMOVL C00213 BC00213 V=400.0  +MOVJ EC00213
SFTON3D P052
SMOVL C00214 BC00214 V=133.3 PL=0  +MOVJ EC00214
SREFP 1 C00215 BC00215  +REFP EC00215
SREFP 2 C00216 BC00216  +REFP EC00216
ARCON
SFTON3D P051
SMOVL C00217 BC00217 V=11.7  +MOVJ EC00217
SMOVL C00218 BC00218 V=11.7  +MOVJ EC00218
SMOVL C00219 BC00219 V=11.7  +MOVJ EC00219
SMOVL C00220 BC00220 V=11.7  +MOVJ EC00220
ARCOF
SMOVL C00221 BC00221 V=166.7  +MOVJ EC00221
SFTOF3D
SMOVL C00222 BC00222 V=400.0  +MOVJ EC00222
SMOVL C00223 BC00223 V=400.0  +MOVJ EC00223
SMOVL C00224 BC00224 V=400.0  +MOVJ EC00224
SMOVL C00225 BC00225 V=400.0  +MOVJ EC00225
SMOVL C00226 BC00226 V=400.0  +MOVJ EC00226
SMOVL C00227 BC00227 V=400.0  +MOVJ EC00227
SMOVL C00228 BC00228 V=400.0  +MOVJ EC00228
SFTON3D P054
SMOVL C00229 BC00229 V=133.3 PL=0  +MOVJ EC00229
ARCON
SMOVL C00230 BC00230 V=11.7  +MOVJ EC00230
SFTON3D P053
SMOVL C00231 BC00231 V=11.7  +MOVJ EC00231
ARCOF
SMOVL C00232 BC00232 V=400.0  +MOVJ EC00232
SFTOF3D
SMOVL C00233 BC00233 V=400.0  +MOVJ EC00233
SMOVL C00234 BC00234 V=400.0  +MOVJ EC00234
SMOVL C00235 BC00235 V=666.7  +MOVJ EC00235
SMOVL C00236 BC00236 V=666.7  +MOVJ EC00236
SMOVL C00237 BC00237 V=400.0  +MOVJ EC00237
SFTON3D P052
SMOVL C00238 BC00238 V=133.3 PL=0  +MOVJ EC00238
ARCON
SMOVL C00239 BC00239 V=11.7  +MOVJ EC00239
SFTON3D P053
SMOVL C00240 BC00240 V=11.7  +MOVJ EC00240
SMOVL C00241 BC00241 V=11.7  +MOVJ EC00241
ARCOF
SMOVL C00242 BC00242 V=166.7  +MOVJ EC00242
SFTOF3D
SMOVL C00243 BC00243 V=400.0  +MOVJ EC00243
SMOVL C00244 BC00244 V=400.0  +MOVJ EC00244
SMOVL C00245 BC00245 V=666.7  +MOVJ EC00245
'Path W1425
SFTOF3D
SFTON3D P023
MOVJ C00246 BC00246 VJ=100.00  +MOVJ EC00246 VJ=100.00
SMOVL C00247 BC00247 V=166.7  +MOVJ EC00247
SMOVL C00248 BC00248 V=133.3 PL=0  +MOVJ EC00248
SREFP 1 C00249 BC00249  +REFP EC00249
SREFP 2 C00250 BC00250  +REFP EC00250
MACRO1 MJ#(0) ARGF14
ARCON
SMOVL C00251 BC00251 V=10.0  +MOVJ EC00251
ARCOF
SMOVL C00252 BC00252 V=400.0  +MOVJ EC00252
SMOVL C00253 BC00253 V=1000.0  +MOVJ EC00253
SFTOF3D
'Path W1426
SFTOF3D
SFTON3D P022
MOVJ C00254 BC00254 VJ=100.00  +MOVJ EC00254 VJ=100.00
SMOVL C00255 BC00255 V=133.3 PL=0  +MOVJ EC00255
SREFP 1 C00256 BC00256  +REFP EC00256
SREFP 2 C00257 BC00257  +REFP EC00257
MACRO1 MJ#(0) ARGF14
ARCON
SMOVL C00258 BC00258 V=10.0  +MOVJ EC00258
ARCOF
SMOVL C00259 BC00259 V=400.0  +MOVJ EC00259
SMOVL C00260 BC00260 V=1000.0  +MOVJ EC00260
SFTOF3D
'Path W1427
SFTOF3D
SFTON3D P021
MOVJ C00261 BC00261 VJ=100.00  +MOVJ EC00261 VJ=100.00
SMOVL C00262 BC00262 V=133.3 PL=0  +MOVJ EC00262
SREFP 1 C00263 BC00263  +REFP EC00263
SREFP 2 C00264 BC00264  +REFP EC00264
MACRO1 MJ#(0) ARGF14
ARCON
SMOVL C00265 BC00265 V=10.0  +MOVJ EC00265
ARCOF
SMOVL C00266 BC00266 V=400.0  +MOVJ EC00266
SFTOF3D
MOVJ C00267 BC00267 VJ=100.00  +MOVJ EC00267 VJ=100.00
MOVJ C00268 BC00268 VJ=100.00  +MOVJ EC00268 VJ=100.00
MOVJ C00269 BC00269 VJ=100.00  +MOVJ EC00269 VJ=100.00
END
